PROGRAM Stn7
VAR

	start7: BOOL;
	reset7: BOOL;

	Stn7ProcessFE: F_TRIG;
	Stn7ProcessRE: R_TRIG;
	bCutStn7ProcessHalt: BOOL;
	DoorClose7: R_TRIG;
	bStn7DoorClamp: BOOL;

END_VAR

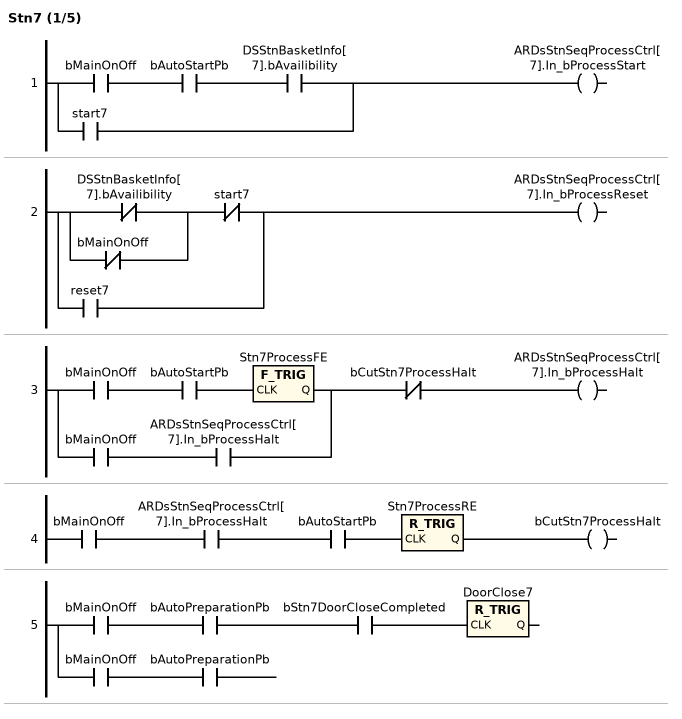
// NETWORK 1
ARDsStnSeqProcessCtrl[7].In_bProcessStart := bMainOnOff AND bAutoStartPb AND DSStnBasketInfo[7].bAvailibility OR start7;

// NETWORK 2
ARDsStnSeqProcessCtrl[7].In_bProcessReset := (NOT DSStnBasketInfo[7].bAvailibility OR NOT bMainOnOff) AND NOT start7 OR reset7;

// NETWORK 3
Stn7ProcessFE(CLK := bMainOnOff AND bAutoStartPb); // F_TRIG
ARDsStnSeqProcessCtrl[7].In_bProcessHalt := (Stn7ProcessFE.Q OR bMainOnOff AND ARDsStnSeqProcessCtrl[7].In_bProcessHalt) AND NOT bCutStn7ProcessHalt;

// NETWORK 4
Stn7ProcessRE(CLK := bMainOnOff AND ARDsStnSeqProcessCtrl[7].In_bProcessHalt AND bAutoStartPb); // R_TRIG
bCutStn7ProcessHalt := Stn7ProcessRE.Q;

// NETWORK 5
DoorClose7(CLK := bMainOnOff AND bAutoPreparationPb AND bStn7DoorCloseCompleted); // R_TRIG
(* DoorClose7.Q OR bMainOnOff AND bAutoPreparationPb; result not used *)

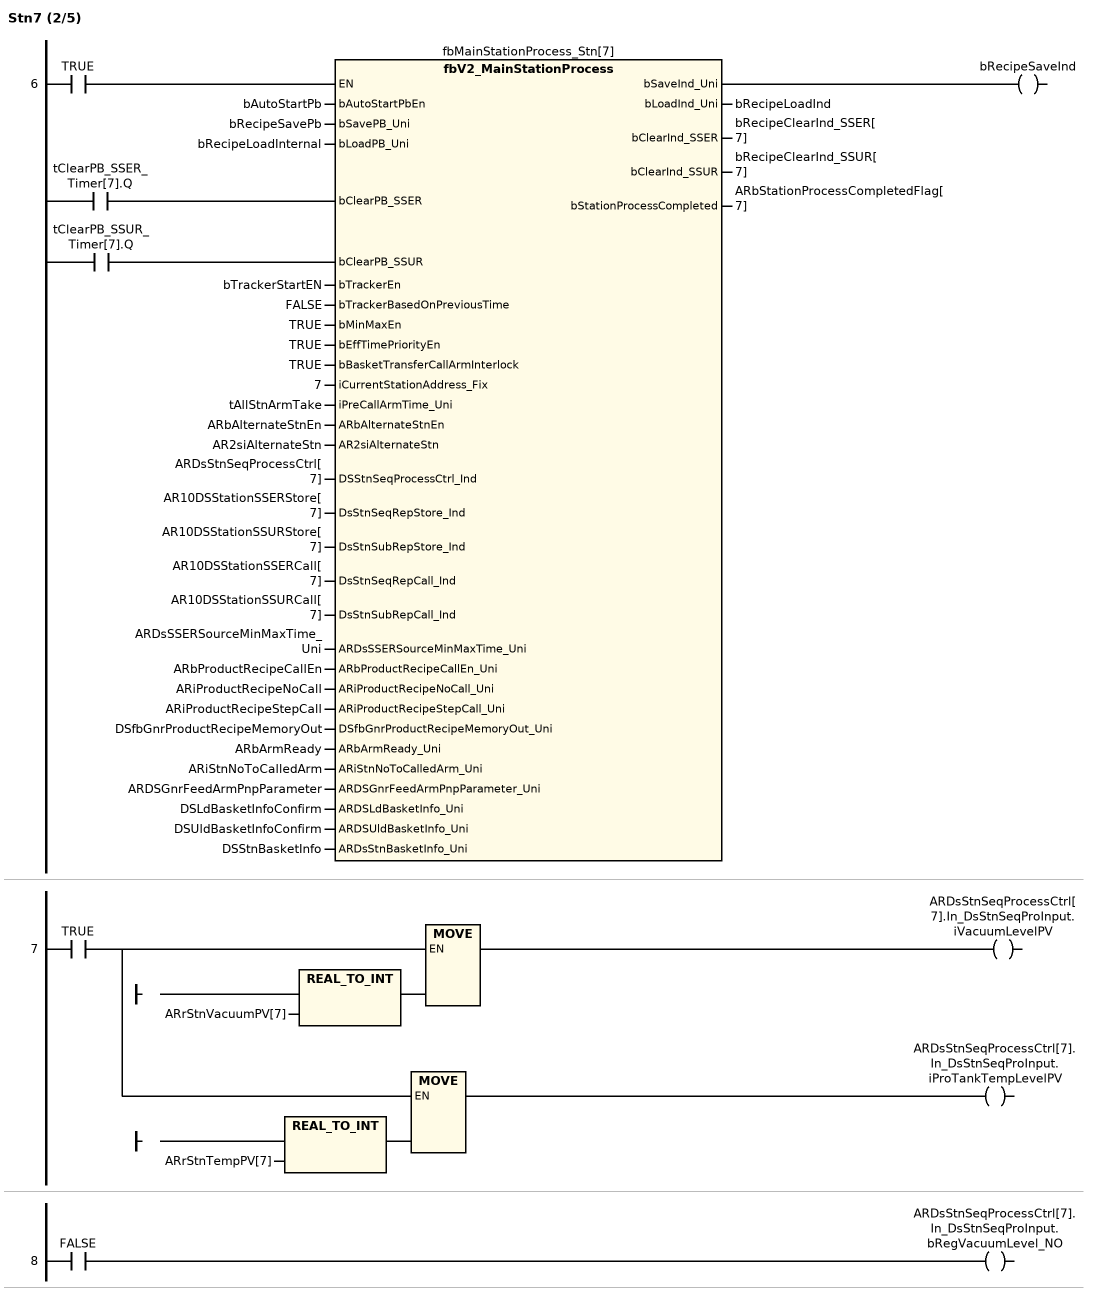
// NETWORK 6
fbMainStationProcess_Stn[7](
    bAutoStartPbEn := bAutoStartPb,
    bSavePB_Uni := bRecipeSavePb,
    bLoadPB_Uni := bRecipeLoadInternal,
    bClearPB_SSER := tClearPB_SSER_Timer[7].Q,
    bClearPB_SSUR := tClearPB_SSUR_Timer[7].Q,
    bTrackerEn := bTrackerStartEN,
    bTrackerBasedOnPreviousTime := FALSE,
    bMinMaxEn := TRUE,
    bEffTimePriorityEn := TRUE,
    bBasketTransferCallArmInterlock := TRUE,
    iCurrentStationAddress_Fix := 7,
    iPreCallArmTime_Uni := tAllStnArmTake,
    ARbAlternateStnEn := ARbAlternateStnEn,
    AR2siAlternateStn := AR2siAlternateStn,
    DSStnSeqProcessCtrl_Ind := ARDsStnSeqProcessCtrl[7],
    DsStnSeqRepStore_Ind := AR10DSStationSSERStore[7],
    DsStnSubRepStore_Ind := AR10DSStationSSURStore[7],
    DsStnSeqRepCall_Ind := AR10DSStationSSERCall[7],
    DsStnSubRepCall_Ind := AR10DSStationSSURCall[7],
    ARDsSSERSourceMinMaxTime_Uni := ARDsSSERSourceMinMaxTime_Uni,
    ARbProductRecipeCallEn_Uni := ARbProductRecipeCallEn,
    ARiProductRecipeNoCall_Uni := ARiProductRecipeNoCall,
    ARiProductRecipeStepCall_Uni := ARiProductRecipeStepCall,
    DSfbGnrProductRecipeMemoryOut_Uni := DSfbGnrProductRecipeMemoryOut,
    ARbArmReady_Uni := ARbArmReady,
    ARiStnNoToCalledArm_Uni := ARiStnNoToCalledArm,
    ARDSGnrFeedArmPnpParameter_Uni := ARDSGnrFeedArmPnpParameter,
    ARDSLdBasketInfo_Uni := DSLdBasketInfoConfirm,
    ARDSUldBasketInfo_Uni := DSUldBasketInfoConfirm,
    ARDsStnBasketInfo_Uni := DSStnBasketInfo,
    bLoadInd_Uni => bRecipeLoadInd,
    bClearInd_SSER => bRecipeClearInd_SSER[7],
    bClearInd_SSUR => bRecipeClearInd_SSUR[7],
    bStationProcessCompleted => ARbStationProcessCompletedFlag[7]); // fbV2_MainStationProcess
bRecipeSaveInd := fbMainStationProcess_Stn[7].bSaveInd_Uni;

// NETWORK 7
ARDsStnSeqProcessCtrl[7].In_DsStnSeqProInput.iVacuumLevelPV := REAL_TO_INT(ARrStnVacuumPV[7]);
ARDsStnSeqProcessCtrl[7].In_DsStnSeqProInput.iProTankTempLevelPV := REAL_TO_INT(ARrStnTempPV[7]);

// NETWORK 8
ARDsStnSeqProcessCtrl[7].In_DsStnSeqProInput.bRegVacuumLevel_NO := FALSE;

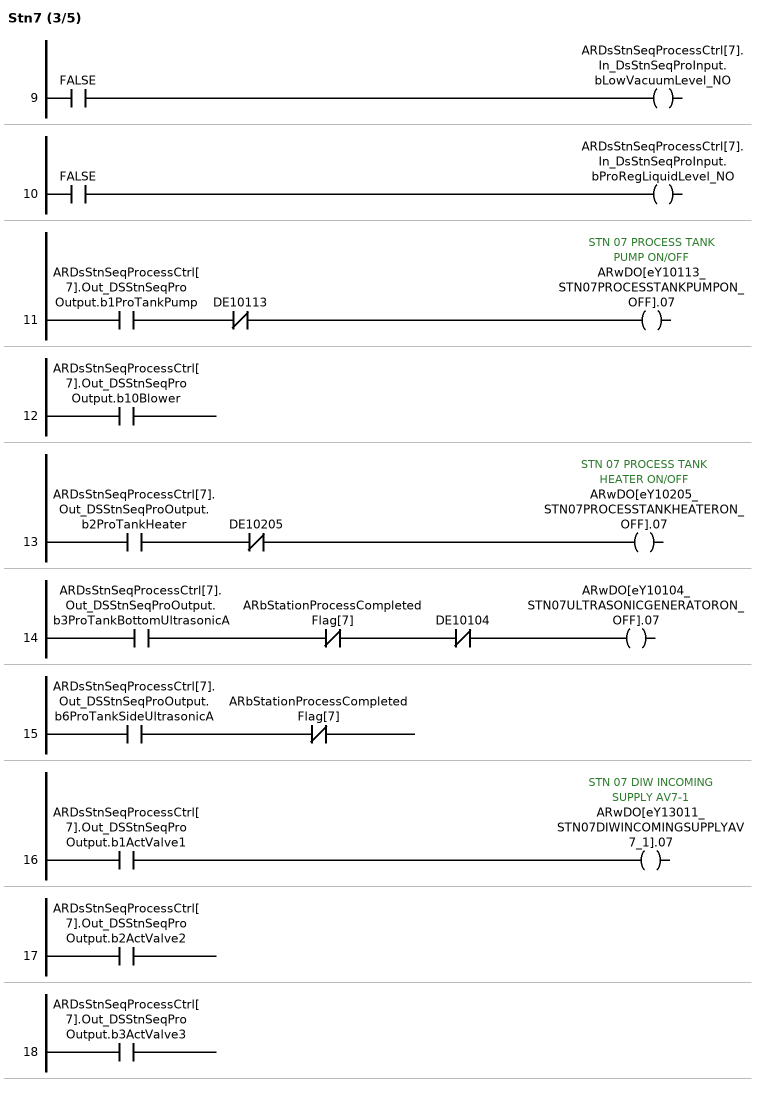
// NETWORK 9
ARDsStnSeqProcessCtrl[7].In_DsStnSeqProInput.bLowVacuumLevel_NO := FALSE;

// NETWORK 10
ARDsStnSeqProcessCtrl[7].In_DsStnSeqProInput.bProRegLiquidLevel_NO := FALSE;

// NETWORK 11
//   ARwDO[eY10113_STN07PROCESSTANKPUMPON_OFF].07: STN 07 PROCESS TANK PUMP ON/OFF
ARwDO[eY10113_STN07PROCESSTANKPUMPON_OFF].07 := ARDsStnSeqProcessCtrl[7].Out_DSStnSeqProOutput.b1ProTankPump AND NOT DE10113;

// NETWORK 12
(* ARDsStnSeqProcessCtrl[7].Out_DSStnSeqProOutput.b10Blower; not connected *)

// NETWORK 13
//   ARwDO[eY10205_STN07PROCESSTANKHEATERON_OFF].07: STN 07 PROCESS TANK HEATER ON/OFF
ARwDO[eY10205_STN07PROCESSTANKHEATERON_OFF].07 := ARDsStnSeqProcessCtrl[7].Out_DSStnSeqProOutput.b2ProTankHeater AND NOT DE10205;

// NETWORK 14
ARwDO[eY10104_STN07ULTRASONICGENERATORON_OFF].07 := ARDsStnSeqProcessCtrl[7].Out_DSStnSeqProOutput.b3ProTankBottomUltrasonicA AND NOT ARbStationProcessCompletedFlag[7] AND NOT DE10104;

// NETWORK 15
(* ARDsStnSeqProcessCtrl[7].Out_DSStnSeqProOutput.b6ProTankSideUltrasonicA AND NOT ARbStationProcessCompletedFlag[7]; result not used *)

// NETWORK 16
//   ARwDO[eY13011_STN07DIWINCOMINGSUPPLYAV7_1].07: STN 07 DIW INCOMING SUPPLY AV7-1
ARwDO[eY13011_STN07DIWINCOMINGSUPPLYAV7_1].07 := ARDsStnSeqProcessCtrl[7].Out_DSStnSeqProOutput.b1ActValve1;

// NETWORK 17
(* ARDsStnSeqProcessCtrl[7].Out_DSStnSeqProOutput.b2ActValve2; not connected *)

// NETWORK 18
(* ARDsStnSeqProcessCtrl[7].Out_DSStnSeqProOutput.b3ActValve3; not connected *)

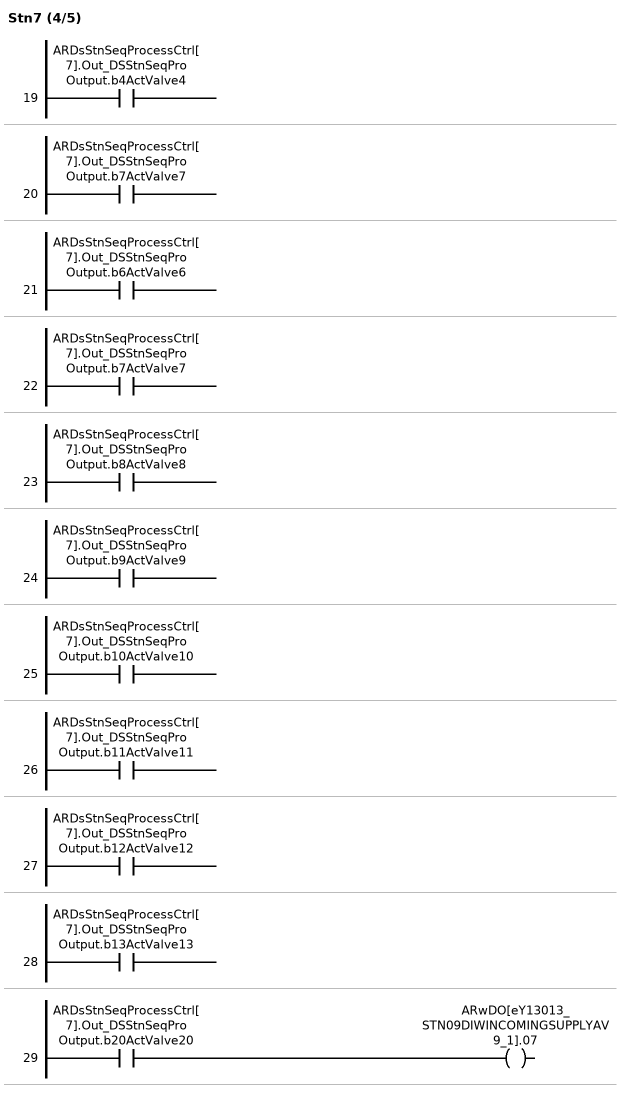
// NETWORK 19
(* ARDsStnSeqProcessCtrl[7].Out_DSStnSeqProOutput.b4ActValve4; not connected *)

// NETWORK 20
(* ARDsStnSeqProcessCtrl[7].Out_DSStnSeqProOutput.b7ActValve7; not connected *)

// NETWORK 21
(* ARDsStnSeqProcessCtrl[7].Out_DSStnSeqProOutput.b6ActValve6; not connected *)

// NETWORK 22
(* ARDsStnSeqProcessCtrl[7].Out_DSStnSeqProOutput.b7ActValve7; not connected *)

// NETWORK 23
(* ARDsStnSeqProcessCtrl[7].Out_DSStnSeqProOutput.b8ActValve8; not connected *)

// NETWORK 24
(* ARDsStnSeqProcessCtrl[7].Out_DSStnSeqProOutput.b9ActValve9; not connected *)

// NETWORK 25
(* ARDsStnSeqProcessCtrl[7].Out_DSStnSeqProOutput.b10ActValve10; not connected *)

// NETWORK 26
(* ARDsStnSeqProcessCtrl[7].Out_DSStnSeqProOutput.b11ActValve11; not connected *)

// NETWORK 27
(* ARDsStnSeqProcessCtrl[7].Out_DSStnSeqProOutput.b12ActValve12; not connected *)

// NETWORK 28
(* ARDsStnSeqProcessCtrl[7].Out_DSStnSeqProOutput.b13ActValve13; not connected *)

// NETWORK 29
ARwDO[eY13013_STN09DIWINCOMINGSUPPLYAV9_1].07 := ARDsStnSeqProcessCtrl[7].Out_DSStnSeqProOutput.b20ActValve20;

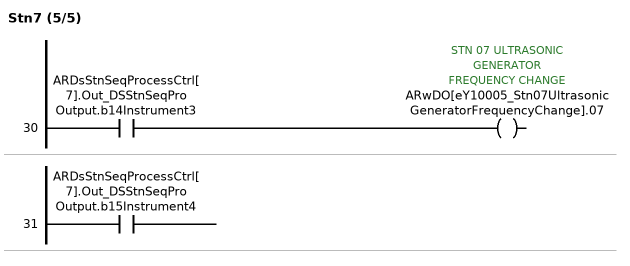
// NETWORK 30
//   ARwDO[eY10005_Stn07UltrasonicGeneratorFrequencyChange].07: STN 07 ULTRASONIC GENERATOR FREQUENCY CHANGE
ARwDO[eY10005_Stn07UltrasonicGeneratorFrequencyChange].07 := ARDsStnSeqProcessCtrl[7].Out_DSStnSeqProOutput.b14Instrument3;

// NETWORK 31
(* ARDsStnSeqProcessCtrl[7].Out_DSStnSeqProOutput.b15Instrument4; not connected *)

END_PROGRAM

(* stored: Version 1.1.0.1, ProductVersion 3.1.4024.12
   POU Stn7: Id {f17301a3-f404-4358-b560-ba8c09013f4e}, SpecialFunc None *)
